(* CoDeSys 2.3 export: N_SYPIALNIA.EXP *)

(* POU Rooms/N_sypialnia, ST *)
FUNCTION_BLOCK N_sypialnia
VAR
	mainLamp:OnOff;
	Shader: ButtonTriggeredShader;
END_VAR
mainLamp(input:=N6_1b, output => N7_1);
shader(input:=N6_1a, shader:=shader_sypialnia, openOut=>N1_1a, closeOut=>N1_1b);
END_FUNCTION_BLOCK
